(* PLC project authorizations, Dassault Systèmes ControlBuild 2024x *)
(* stored: creationDateTime 2023-10-03T11:13:50-01:00 *)

FUNCTION_BLOCK tni_train.authorizations
  VAR_INPUT
    AuthorizationClosingLeftC1 : BOOL := false;
    AuthorizationOpeningRightC1 : BOOL := false;
    AuthorizationClosingRightC1 : BOOL := false;
    AuthorizationOpeningLeftC1 : BOOL := false;
  END_VAR
  VAR_INPUT
    AuthorizationClosingLeftC2 : BOOL := false;
    AuthorizationOpeningRightC2 : BOOL := false;
    AuthorizationClosingRightC2 : BOOL := false;
    AuthorizationOpeningLeftC2 : BOOL := false;
  END_VAR
  VAR_OUTPUT
    AuthorizationOpeningLeft : BOOL := false;
    AuthorizationClosingLeft : BOOL := false;
  END_VAR
  VAR_OUTPUT
    AuthorizationOpeningRight : BOOL := false;
    AuthorizationClosingRight : BOOL := false;
  END_VAR

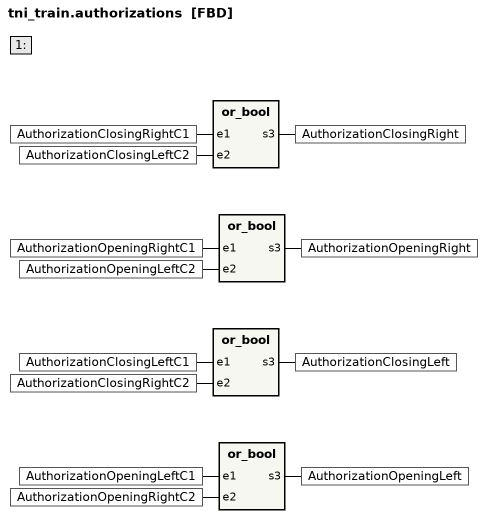
(* FBD diagram, written out as Structured Text *)
1:
AuthorizationClosingRight := or_bool(AuthorizationClosingRightC1, AuthorizationClosingLeftC2);
AuthorizationOpeningRight := or_bool(AuthorizationOpeningRightC1, AuthorizationOpeningLeftC2);
AuthorizationClosingLeft := or_bool(AuthorizationClosingLeftC1, AuthorizationClosingRightC2);
AuthorizationOpeningLeft := or_bool(AuthorizationOpeningLeftC1, AuthorizationOpeningRightC2);
END_FUNCTION_BLOCK
